Universal Robots PolyScope program: rtde_control_loop.urp

Program rtde_control_loop_guillermo (installation=default directory=/programs/usbdisk createdIn=3.2.19275.0 lastSavedIn=5.5.1.82186 robotSerialNumber=20185000228)
Calibrated DH parameters: a=[-0.000126, -0.253171, -0.571397, -0.00001, -0.000004, 0]; d=[0.180809, 253.684169, -261.31341, 7.803768, 0.119899, 0.115655]; alpha=[1.570233, -0.0022, -0.002379, 1.571202, -1.570947, 0]; deltaTheta=[0, -1.14496, 7.459905, -0.03176, -0.000002, 0]
BeforeStart
  setp := Joint_6_name
  SuppressedNode
    Script: rtde_set_watchdog("input_int_register_0", 1, "PAUSE")
Robot Program (runOnlyOnce=false)
  Script: write_output_integer_register(0, 0)
  Script: sync()
  SuppressedNode
    MoveL speed 250 mm/s, acceleration 1200 mm/s^2 (useActiveTCP=true) feature=Base
      Waypoint Waypoint (Variable): variable=setp
  Loop Forever
    Script: servoj(get_inverse_kin(setp),0,0,0.25,0.2,1000)
  Script: write_output_integer_register(0, 1)
  Script: sync()
Thread Thread_1 (runOnlyOnce=false)
  setp := Joint_6_name
  Loop Forever
    tmp := p[0,0,0,0,0,0]
    Script: tmp[0] = read_input_float_register(0)
    Script: tmp[1] = read_input_float_register(1)
    Script: tmp[2] = read_input_float_register(2)
    Script: tmp[3] = read_input_float_register(3)
    Script: tmp[4] = read_input_float_register(4)
    Script: tmp[5] = read_input_float_register(5)
    If tmp != p[0,0,0,0,0,0]
      setp := tmp
    var_1 := get_actual_tcp_speed()
    var_2 := norm([var_1[0],var_1[1],var_1[2]])
    Script: sync()
